ABB RobotStudio station: Practica3.rspag

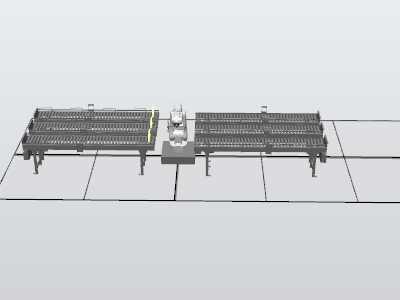
--- station ---
Station Practica3 (saved by RobotStudio 25.4.11475.0)
Controller IRB120_3_58
  mechanical unit ROB_1: IRB120_3_58__01, 6 joints, base frame (0, 0, 0) mm
Layout (positions relative to the parent item):
  - IRB120_3_58__01 [mechanism, from %ABB.RobotStudio.Models.IRB120%\IRB120_3_58_G_01.rslib] at (0, 0, 0) mm; joint values [0, 0, 0, 0, 0.5236, 0] (rad or m)
  - MyNewTool [mechanism] at (364.35, 0, 594) mm, rotated rx -150 ry 0 rz 90 deg
      TCP Centro at (0, 0, 0) mm, rotated rx -90 ry 0 rz 90 deg
      TCP Ventosas3 at (0, 0, -95) mm, rotated rx -90 ry 0 rz 90 deg
      TCP Ventosas4 at (0, 0, 95) mm, rotated rx -90 ry 0 rz 90 deg
      links: Enganche_4
  - Peana [part] at (-200, -200, 0) mm, size 400 x 400 x 100 mm
  - Cinta1 [part] at (-211.15, -1753.75, 0) mm, rotated rx 0 ry 0 rz 90 deg, size 1516.5 x 295 x 472.5 mm
  - Cinta4 [part] at (-387.39, 1694.43, 0) mm, rotated rx 0 ry 0 rz -90 deg, size 1516.5 x 295 x 472.5 mm
  - Cinta2 [part] at (105.68, -1750.96, 0) mm, rotated rx 0 ry 0 rz 90 deg, size 1516.5 x 295 x 472.5 mm
  - Cinta3 [part] at (438.1, -1753.58, 0) mm, rotated rx 0 ry 0 rz 90 deg, size 1516.5 x 295 x 472.5 mm
  - Cinta6 [part] at (250.29, 1696.68, 0) mm, rotated rx 0 ry 0 rz -90 deg, size 1516.5 x 295 x 472.5 mm
  - Cinta5 [part] at (-84.57, 1695.15, 0) mm, rotated rx 0 ry 0 rz -90 deg, size 1516.5 x 295 x 472.5 mm
  - Caja_Tipo1 [part] at (-366, -1693, 382) mm, size 100 x 100 x 50 mm
  - Caja_Tipo2 [part] at (-37, -1686.06, 382.65) mm, size 100 x 100 x 80 mm
  - Caja_Tipo3 [part] at (290, -1683, 388) mm, size 100 x 100 x 100 mm
  - SC_Cinta1 [smart component]
      signals: DI DI_Gen_T1, DI DI_Gen_T2, DI DI_Gen_T3, DO DO_Sensor_Bajo, DO DO_Sensor_Medio, DO DO_Sensor_Alto, DI DI_Mover_C1
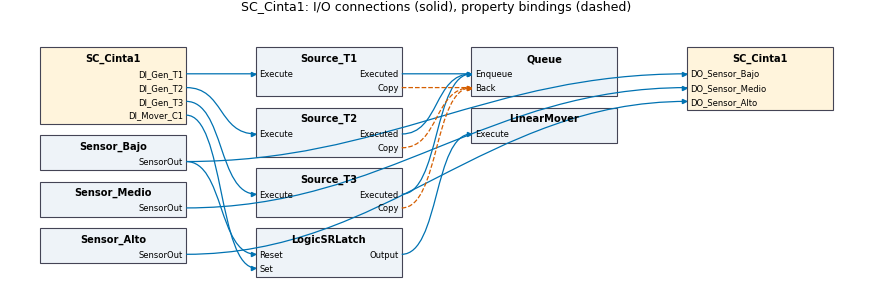
      connections:
        SC_Cinta1.DI_Gen_T1 -> Source_T1.Execute
        SC_Cinta1.DI_Gen_T2 -> Source_T2.Execute
        SC_Cinta1.DI_Gen_T3 -> Source_T3.Execute
        Source_T1.Executed -> Queue.Enqueue
        Source_T2.Executed -> Queue.Enqueue
        Source_T3.Executed -> Queue.Enqueue
        Sensor_Bajo.SensorOut -> SC_Cinta1.DO_Sensor_Bajo
        Sensor_Medio.SensorOut -> SC_Cinta1.DO_Sensor_Medio
        Sensor_Alto.SensorOut -> SC_Cinta1.DO_Sensor_Alto
        Sensor_Bajo.SensorOut -> LogicSRLatch.Reset
        LogicSRLatch.Output -> LinearMover.Execute
        SC_Cinta1.DI_Mover_C1 -> LogicSRLatch.Set
        Source_T1.Copy => Queue.Back
        Source_T2.Copy => Queue.Back
        Source_T3.Copy => Queue.Back
    - Source_T1 [smart component, from Components\Source.rslib] at (0, 878.4, 0) mm
        properties: Source=Caja_Tipo1; Copy=(none); Parent=(none); Position=[-0.366 -1.693 0.382]; Orientation=[0 0 0]; Transient=false; PhysicsBehavior=-1
    - Source_T2 [smart component, from Components\Source.rslib]
        properties: Source=Caja_Tipo2; Copy=(none); Parent=(none); Position=[-0.366 -1.693 0.382]; Orientation=[0 0 0]; Transient=false; PhysicsBehavior=-1
    - Source_T3 [smart component, from Components\Source.rslib]
        properties: Source=Caja_Tipo3; Copy=(none); Parent=(none); Position=[-0.366 -1.693 0.382]; Orientation=[0 0 0]; Transient=false; PhysicsBehavior=-1
    - Queue [smart component, from Components\Queue.rslib]
        properties: Back=(none); Front=(none); Queue={ae4d30b3-6302-4111-9fee-83a94bcd6a61};{9fa5510e-041f-4493-96ec-c95941a7de32};{5319e2fc-a695-4427-a68f-7cbe0e69f7e4};{3efef574-f5d8-49aa-a5b4-01e6362c16f4};{a1e64e2e-bae4-4094-9af5-35717dc52df0};{90407918-cd8a-43af-9253-99db0ca8b2cd};{5acc8fc2-0798-4915-81ff-b25f6d5593ec};{61423d0f-f941-4e73-af3b-112a04a09b53};{953f87a9-bdd4-4cb4-a80c-3d35c462e832};{1631f3d6-8d09-4da0-8cec-8cbaa0fb8792};{cab1151d-17ff-416b-9bb8-76c1a92ffb11};{709a4bb6-f8ae-485e-a46f-52f42bc28a03};{757c1d3f-b98b-4062-b6e4-9dd61a946051};{b9655f3a-bf60-4423-91ba-6a07460e28c4};{d7396197-064d-4214-b519-df7028a49eeb};{af7f2dd8-8d2d-49ce-bc3f-f1ae0ce77ebb};{56c8aa57-b622-4854-bfd4-cc37ea0eaac4};{93e1c836-db4d-4383-b321-3c540578f93f};{c1cab4d0-5605-4614-acff-7234784f2794};{21a5687b-13b3-45a7-a44d-9ef329473538};{e8432f60-373c-4531-8b0a-4d6747e82efe};{1b8eaf30-fe4c-4f09-99cb-c14138031cc8};{9ef8b087-f2a4-45a1-916a-8d388a000a67};{ac3eefbd-dbbd-4806-b8d9-2bdfa1e66709};{6bbb20f7-4848-4c6b-80bb-41a8ed0c3422};{560186ce-d231-4b2f-9cb0-d667fd014fff};{8ef24d2c-7559-482c-9b53-3d872e96b759};{638ee7c7-692f-400c-862d-77c483a76bbb};{18bf07ff-95d7-44c5-ac93-6077ee389aad};{a14bbcad-93fe-4a17-8c33-dc9a6455d2bc};{1956f7e1-81a8-4c4b-a953-4b234403df65};{055c1d69-0d71-46b2-a09d-feb5f3c0ad83};{6400679a-db5a-4c21-bd62-84ae49f8a382};{37c3a838-eb8e-4eb3-96b1-78701e28feef};{289cf7f1-5e36-4ccd-ab18-b29cd6d78d4d};{62f60689-158a-485b-9bfe-8d9deff740b5};{17fe60c0-212e-4ef7-aef1-3c5e78d04126};{c8c3b35f-117b-4ef3-ac39-44fc0f9ecd59};{6bfb9224-18d2-413a-84f5-a1e35e777d4f};{ea2980e8-0bc9-4d52-a2a1-1e1a2d485450};{6993df89-24a9-4713-b949-d7ca80afb984};{2c206039-b06b-44be-9fb2-e4e3ab796f06};{47dba929-5f9b-4cf8-b146-fed9fac773aa};{4920f1fd-ca38-4464-85c7-93d89a30eeed}; NumberOfObjects=2
    - LinearMover [smart component, from Components\LinearMover.rslib]
        properties: Object=Queue; Direction=[0 0.001 0]; Speed=0.15; Reference=Global; ReferenceObject=(none)
    - Sensor_Bajo [smart component, from Components\LineSensor.rslib]
        properties: Start=[-0.411 -0.319 0.42]; End=[-0.21 -0.319 0.42]; Length=0.201; Radius=0; Tag=(none); SenseMultiple=false; SensedPart=(none); SensedPoint=[0 0 0]
      - _sensorPart_ [part], size 201 x 0 x 0 mm
    - Sensor_Medio [smart component, from Components\LineSensor.rslib]
        properties: Start=[-0.411 -0.319 0.46]; End=[-0.21 -0.319 0.46]; Length=0.201; Radius=0; Tag=(none); SenseMultiple=false; SensedPart=(none); SensedPoint=[0 0 0]
      - _sensorPart_ [part], size 201 x 0 x 0 mm
    - Sensor_Alto [smart component, from Components\LineSensor.rslib]
        properties: Start=[-0.411 -0.319 0.48]; End=[-0.21 -0.319 0.48]; Length=0.201; Radius=0; Tag=(none); SenseMultiple=false; SensedPart=(none); SensedPoint=[0 0 0]
      - _sensorPart_ [part], size 201 x 0 x 0 mm
    - LogicSRLatch [smart component, from Components\LogicSRLatch.rslib]
  - SC_Cinta2 [smart component]
      signals: DI DI_Mover_C2, DI DI_Gen_C1, DI DI_Gen_C2, DI DI_Gen_C3, DO DO_Sensor_Bajo, DO DO_Sensor_Medio, DO DO_Sensor_Alto
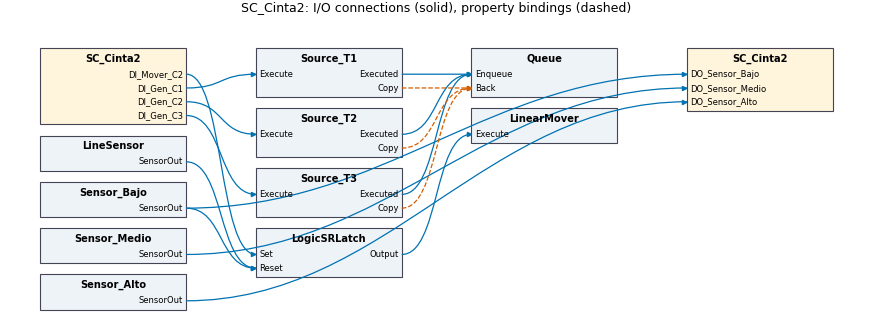
      connections:
        SC_Cinta2.DI_Mover_C2 -> LogicSRLatch.Set
        SC_Cinta2.DI_Gen_C1 -> Source_T1.Execute
        SC_Cinta2.DI_Gen_C2 -> Source_T2.Execute
        SC_Cinta2.DI_Gen_C3 -> Source_T3.Execute
        Source_T1.Executed -> Queue.Enqueue
        Source_T2.Executed -> Queue.Enqueue
        Source_T3.Executed -> Queue.Enqueue
        LogicSRLatch.Output -> LinearMover.Execute
        LineSensor.SensorOut -> LogicSRLatch.Reset
        Sensor_Bajo.SensorOut -> LogicSRLatch.Reset
        Sensor_Bajo.SensorOut -> SC_Cinta2.DO_Sensor_Bajo
        Sensor_Medio.SensorOut -> SC_Cinta2.DO_Sensor_Medio
        Sensor_Alto.SensorOut -> SC_Cinta2.DO_Sensor_Alto
        Source_T3.Copy => Queue.Back
        Source_T2.Copy => Queue.Back
        Source_T1.Copy => Queue.Back
    - LinearMover [smart component, from Components\LinearMover.rslib]
        properties: Object=Queue; Direction=[0 0.001 0]; Speed=0.15; Reference=Global; ReferenceObject=(none)
    - LogicSRLatch [smart component, from Components\LogicSRLatch.rslib]
    - Source_T2 [smart component, from Components\Source.rslib] at (0, 878.4, 0) mm
        properties: Source=Caja_Tipo2; Copy=(none); Parent=(none); Position=[-0.037 -1.683 0.388]; Orientation=[0 0 0]; Transient=false; PhysicsBehavior=-1
    - Source_T3 [smart component, from Components\Source.rslib] at (0, 878.4, 0) mm
        properties: Source=Caja_Tipo3; Copy=(none); Parent=(none); Position=[-0.037 -1.683 0.388]; Orientation=[0 0 0]; Transient=false; PhysicsBehavior=-1
    - Source_T1 [smart component, from Components\Source.rslib] at (0, 878.4, 0) mm
        properties: Source=Caja_Tipo1; Copy=(none); Parent=(none); Position=[-0.037 -1.683 0.388]; Orientation=[0 0 0]; Transient=false; PhysicsBehavior=-1
    - Queue [smart component, from Components\Queue.rslib]
        properties: Back=(none); Front=(none); Queue={2bcd5c23-c1ed-46e9-8c09-8f83fa8b4f7f};{6c76dee3-31f3-442e-bd1e-8fd0cd5ca1d8};{87979af6-ae82-445d-8c1c-a2b879dac4d6};{eee5c5c7-d8e7-4388-a9cb-2509ca800b36};{0ed9a9c4-d81e-4250-8c3f-7bd06b761d9a};{48cb68ef-0ffe-479b-be93-44ded6a24c72};{ede27b09-c003-47f3-a151-95e2712a7b0c};{a391c974-7157-4c51-ac27-7ab25ebc9bf4};{96269cb6-2ddd-45c1-a0d0-c3bba03121e4};{308577e6-806f-4c99-832e-8584b715af30};{7a8da34a-d222-4c7e-9417-0fb4f6fe10c3};{51fd84be-2d47-4bb8-9c48-63eea8f1a314};{4f8447d2-d18b-4198-b70f-0fde71820eac};{26466b57-75da-4393-8d5b-4afc74e56a4b};{388f5636-77e2-470e-ac11-c912e79f43ad};{6e4eb306-18d5-49c2-bef4-ace6f9cce639};{bbdeb09b-5027-4537-9290-c9dec0b41319};{d1ec0450-83df-4b2e-a66f-ffe360aa7048};{c7e78e88-61bb-4ac1-b0f7-c37af5dace11};{622ee8d1-b9ad-42ff-9941-53bfff9b80b7};{5b86faa8-1afa-4e94-a375-27763fc04b84};{0319b542-081c-49c6-b7df-58ec952c4440}; NumberOfObjects=2
    - Sensor_Bajo [smart component, from Components\LineSensor.rslib]
        properties: Start=[-0.085 -0.319 0.42]; End=[0.09 -0.319 0.42]; Length=0.175; Radius=0; Tag=(none); SenseMultiple=false; SensedPart=(none); SensedPoint=[0 0 0]
      - _sensorPart_ [part], size 175 x 0 x 0 mm
    - Sensor_Medio [smart component, from Components\LineSensor.rslib]
        properties: Start=[-0.085 -0.319 0.46]; End=[0.09 -0.319 0.46]; Length=0.175; Radius=0; Tag=(none); SenseMultiple=false; SensedPart=(none); SensedPoint=[0 0 0]
      - _sensorPart_ [part], size 175 x 0 x 0 mm
    - Sensor_Alto [smart component, from Components\LineSensor.rslib]
        properties: Start=[-0.085 -0.319 0.48]; End=[0.09 -0.319 0.48]; Length=0.175; Radius=0; Tag=(none); SenseMultiple=false; SensedPart=(none); SensedPoint=[0 0 0]
      - _sensorPart_ [part], size 175 x 0 x 0 mm
  - SC_Cinta3 [smart component]
      signals: DI DI_Gen_T1, DI DI_Gen_T2, DI DI_Gen_T3, DO DO_Sensor_Bajo, DO DO_Sensor_Medio, DO DO_Sensor_Alto, DI DI_Mover_C3
      connections:
        LogicSRLatch_3.Output -> LinearMover_2.Execute
        Source_T1.Executed -> Queue_2.Enqueue
        Source_T2.Executed -> Queue_2.Enqueue
        Source_T3.Executed -> Queue_2.Enqueue
        SC_Cinta3.DI_Gen_T1 -> Source_T1.Execute
        SC_Cinta3.DI_Gen_T2 -> Source_T2.Execute
        SC_Cinta3.DI_Gen_T3 -> Source_T3.Execute
        Sensor_Bajo.SensorOut -> SC_Cinta3.DO_Sensor_Bajo
        Sensor_Bajo.SensorOut -> LogicSRLatch_3.Reset
        Sensor_Medio.SensorOut -> SC_Cinta3.DO_Sensor_Medio
        Sensor_Alto.SensorOut -> SC_Cinta3.DO_Sensor_Alto
        SC_Cinta3.DI_Mover_C3 -> LogicSRLatch_3.Set
        Source_T1.Copy => Queue_2.Back
        Source_T2.Copy => Queue_2.Back
        Source_T3.Copy => Queue_2.Back
    - Source_T1 [smart component, from Components\Source.rslib]
        properties: Source=Caja_Tipo1; Copy=(none); Parent=(none); Position=[0.29 -1.683 0.388]; Orientation=[0 0 0]; Transient=false; PhysicsBehavior=-1
    - Sensor_Bajo [smart component, from Components\LineSensor.rslib]
        properties: Start=[0.237 -0.319 0.42]; End=[0.438 -0.319 0.42]; Length=0.201; Radius=0; Tag=(none); SenseMultiple=false; SensedPart=(none); SensedPoint=[0 0 0]
      - _sensorPart_ [part], size 201 x 0 x 0 mm
    - Queue_2 [smart component, from Components\Queue.rslib]
        properties: Back=(none); Front=(none); Queue={b5c0da53-b886-4eab-a8f7-240ca8277bb4};{162bf9dd-af30-44ee-bf84-297d0a330099};{1ce0c98b-bb50-4a90-8f2b-f630c16990df};{7d84dcbd-445a-4615-af1b-5e8ef1b0da41};{f2ce0fef-d506-4055-bce7-edc570f5b85d};{49ed6fa6-4484-4528-a036-6e04abb92bae};{51e9f9c3-66fc-43a1-92ef-84e0ce0dd9ee};{a6f4487b-d18e-4f28-a26b-d157c1f4e47e};{40463528-f2a5-4b0f-801e-c86bb77c77c6};{7bbab9be-23ff-4f72-bedf-08c0365cb3c3};{96a9fc0c-d42f-4625-b4ce-ff104d0d23d5};{38a37ed4-7e6c-411f-af4e-19aff20a759d};{77cec95b-3a46-431e-99ce-bad3b8b5176a};{a7fffe4b-cb80-4798-9ffc-81a953cfccc9};{07ba421a-4e5e-4a4c-8141-2298dd789c99};{14acecfe-8c89-4afa-883c-57a0848518f5};{03d718bc-ab0b-4980-ad5a-f10c83bcab31};{af4d491e-c72f-4645-8bd7-c3d7c8b11cec};{0fcde2d3-d7fc-49db-9a2c-edd93dbc6e02};{0f9b7fda-dccf-447b-aa29-b1cebfc17353};{32b10893-1c7e-43b2-a21f-2af3cf555bbd};{ef222544-086f-4277-904e-25c3415c13a1};{819d3b9b-c1dd-4f60-9c29-6154756c0372};{19730fc8-a8c3-4879-83ee-9a8b8ef66b87};{472fec01-8044-440c-8fff-ca474cbc4876};{4a0d8dfd-107d-4185-9536-f8a48dfdc9b6};{2941b239-3e65-4e98-8b67-6c5e40cb0733}; NumberOfObjects=1
    - LinearMover_2 [smart component, from Components\LinearMover.rslib]
        properties: Object=Queue_2; Direction=[0 0.001 0]; Speed=0.15; Reference=Global; ReferenceObject=(none)
    - LogicSRLatch_3 [smart component, from Components\LogicSRLatch.rslib]
    - Source_T2 [smart component, from Components\Source.rslib]
        properties: Source=Caja_Tipo2; Copy=(none); Parent=(none); Position=[0.29 -1.683 0.388]; Orientation=[0 0 0]; Transient=false; PhysicsBehavior=-1
    - Source_T3 [smart component, from Components\Source.rslib]
        properties: Source=Caja_Tipo3; Copy=(none); Parent=(none); Position=[0.29 -1.683 0.388]; Orientation=[0 0 0]; Transient=false; PhysicsBehavior=-1
    - Sensor_Medio [smart component, from Components\LineSensor.rslib]
        properties: Start=[0.237 -0.319 0.46]; End=[0.438 -0.319 0.46]; Length=0.201; Radius=0; Tag=(none); SenseMultiple=false; SensedPart=(none); SensedPoint=[0 0 0]
      - _sensorPart_ [part], size 201 x 0 x 0 mm
    - Sensor_Alto [smart component, from Components\LineSensor.rslib]
        properties: Start=[0.237 -0.319 0.48]; End=[0.438 -0.319 0.48]; Length=0.201; Radius=0; Tag=(none); SenseMultiple=false; SensedPart=(none); SensedPoint=[0 0 0]
      - _sensorPart_ [part], size 201 x 0 x 0 mm
  - SC_Agarre [smart component]
      connections:
        LogicGate.Output -> Detacher.Execute
        CollisionSensor_2.SensorOut -> Detacher.Execute
        CollisionSensor.SensorOut -> Attacher.Execute
        CollisionSensor_3.SensorOut -> Attacher_2.Execute
        CollisionSensor_4.SensorOut -> Detacher_2.Execute
        CollisionSensor_2.SensorOut -> Detacher_2.Execute
        CollisionSensor.Part2 => Attacher.Child
        CollisionSensor.Part2 => Detacher.Child
        CollisionSensor_3.Part2 => Attacher_2.Child
        CollisionSensor_3.Part2 => Detacher.Child
    - Attacher [smart component, from Components\Attacher.rslib]
        properties: Parent=MyNewTool; Flange=1; Child=(none); Mount=false; Offset=[0 0 0]; Orientation=[0 0 0]
    - Detacher [smart component, from Components\Detacher.rslib]
        properties: Child=(none); KeepPosition=true
    - CollisionSensor [smart component, from Components\CollisionSensor.rslib]
        properties: Object1=MyNewTool; Object2=(none); NearMiss=0; Part1=(none); Part2=(none); CollisionType=0
    - CollisionSensor_2 [smart component, from Components\CollisionSensor.rslib]
        properties: Object1=MyNewTool; Object2=Grupo_1; NearMiss=0; Part1=(none); Part2=(none); CollisionType=0
    - CollisionSensor_3 [smart component, from Components\CollisionSensor.rslib]
        properties: Object1=MyNewTool; Object2=(none); NearMiss=0; Part1=(none); Part2=(none); CollisionType=0
    - Attacher_2 [smart component, from Components\Attacher.rslib]
        properties: Parent=MyNewTool; Flange=2; Child=(none); Mount=false; Offset=[0 0 0]; Orientation=[0 0 0]
  - Grupo_1 [graphiccomponentgroup]
    - Caja [part] at (-339.08, 251.28, 364.37) mm, size 100 x 100 x 50 mm
    - Caja_2 [part] at (-37, 355.02, 378.78) mm, size 100 x 100 x 80 mm
    - Pieza_1 [part] at (37.54, -45.56, 52.42) mm, size 100 x 100 x 100 mm
Attachment: MyNewTool is attached to IRB120_3_58__01 / Link6
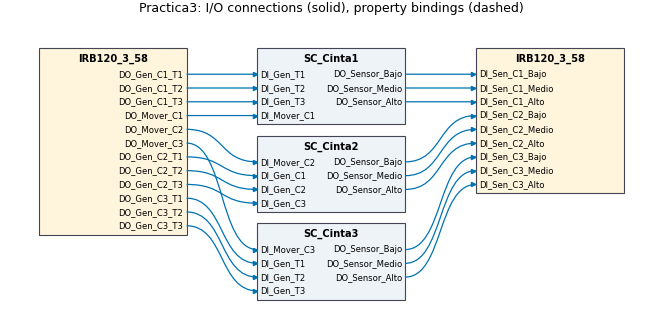
Station logic (signal -> signal, property => property):
  IRB120_3_58.DO_Gen_C1_T1 -> SC_Cinta1.DI_Gen_T1
  IRB120_3_58.DO_Gen_C1_T2 -> SC_Cinta1.DI_Gen_T2
  IRB120_3_58.DO_Gen_C1_T3 -> SC_Cinta1.DI_Gen_T3
  SC_Cinta1.DO_Sensor_Bajo -> IRB120_3_58.DI_Sen_C1_Bajo
  SC_Cinta1.DO_Sensor_Medio -> IRB120_3_58.DI_Sen_C1_Medio
  SC_Cinta1.DO_Sensor_Alto -> IRB120_3_58.DI_Sen_C1_Alto
  IRB120_3_58.DO_Mover_C1 -> SC_Cinta1.DI_Mover_C1
  IRB120_3_58.DO_Mover_C2 -> SC_Cinta2.DI_Mover_C2
  IRB120_3_58.DO_Mover_C3 -> SC_Cinta3.DI_Mover_C3
  SC_Cinta2.DO_Sensor_Bajo -> IRB120_3_58.DI_Sen_C2_Bajo
  SC_Cinta2.DO_Sensor_Medio -> IRB120_3_58.DI_Sen_C2_Medio
  SC_Cinta2.DO_Sensor_Alto -> IRB120_3_58.DI_Sen_C2_Alto
  SC_Cinta3.DO_Sensor_Bajo -> IRB120_3_58.DI_Sen_C3_Bajo
  SC_Cinta3.DO_Sensor_Medio -> IRB120_3_58.DI_Sen_C3_Medio
  SC_Cinta3.DO_Sensor_Alto -> IRB120_3_58.DI_Sen_C3_Alto
  IRB120_3_58.DO_Gen_C2_T1 -> SC_Cinta2.DI_Gen_C1
  IRB120_3_58.DO_Gen_C2_T2 -> SC_Cinta2.DI_Gen_C2
  IRB120_3_58.DO_Gen_C2_T3 -> SC_Cinta2.DI_Gen_C3
  IRB120_3_58.DO_Gen_C3_T1 -> SC_Cinta3.DI_Gen_T1
  IRB120_3_58.DO_Gen_C3_T2 -> SC_Cinta3.DI_Gen_T2
  IRB120_3_58.DO_Gen_C3_T3 -> SC_Cinta3.DI_Gen_T3

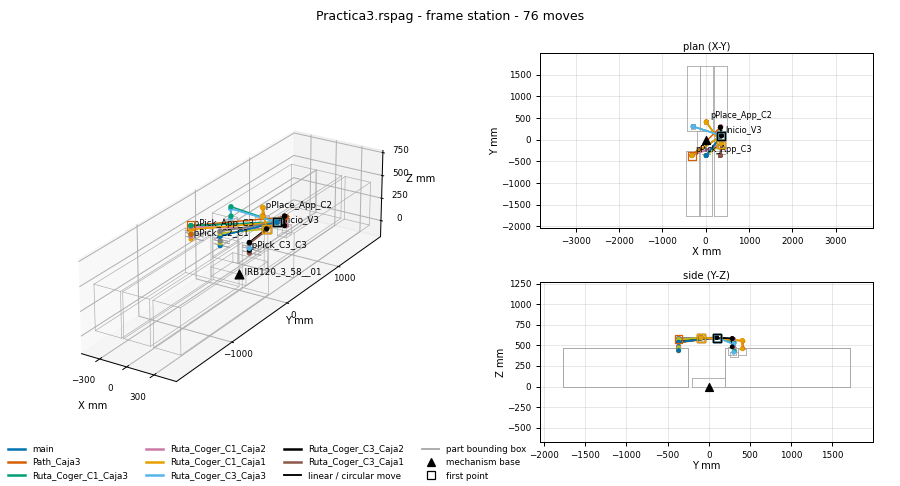
[picture p0: tool path of Practica3.rspag in frame station, 76 of 76 moves have a stored position in this frame; points joined in program order, loops and branches not executed]
--- Controller Data/IRB120_3_58/RAPID/TASK1/PROGMOD/CalibData.mod ---
MODULE CalibData
    PERS tooldata Centro:=[TRUE,[[0,0,0],[1,0,0,0]],[1,[0,0,1],[1,0,0,0],0,0,0]];
    PERS tooldata Ventosas3:=[TRUE,[[0,95,0],[1,0,0,0]],[1,[0,0,1],[1,0,0,0],0,0,0]];
    PERS tooldata Ventosas4:=[TRUE,[[0,-95,0],[1,0,0,0]],[1,[0,0,1],[1,0,0,0],0,0,0]];
ENDMODULE

--- Controller Data/IRB120_3_58/RAPID/TASK1/PROGMOD/Module1.mod ---
MODULE Module1


    CONST robtarget pPick_App_C3:=[[-316,-368.6,572],[0,0,-0.707106781,0.707106781],[-2,0,-2,0],[9E+09,9E+09,9E+09,9E+09,9E+09,9E+09]];
    CONST robtarget pPick_C3_C_1:=[[-316,-368.6,482],[0,0,-0.707106781,0.707106781],[-2,1,-3,0],[9E+09,9E+09,9E+09,9E+09,9E+09,9E+09]];
    CONST robtarget pPlace_App_C6:=[[349.296,299.975,572],[0.5,-0.5,0.5,-0.5],[0,-1,-1,0],[9E+09,9E+09,9E+09,9E+09,9E+09,9E+09]];
    CONST robtarget pPlace_C3_C_6:=[[349.296,299.975,482],[0.5,-0.5,0.5,-0.5],[0,-2,0,0],[9E+09,9E+09,9E+09,9E+09,9E+09,9E+09]];
    CONST robtarget Inicio_V3:=[[364.353821314,95.000001192,593.99994615],[0.499999995,0,0.866025407,0],[-1,0,-1,0],[9E+09,9E+09,9E+09,9E+09,9E+09,9E+09]];

    ! Variables para la generacion aleatoria
    VAR num nCintaAleatoria := 0;
    VAR num nTipoAleatorio := 0;
    VAR num nSeed := 42;

    ! Contadores y requeridas
    VAR num nCajasT1_Req := 0;
    VAR num nCajasT2_Req := 0;
    VAR num nCajasT3_Req := 0;
    VAR num nCajasT1_Gen := 0;
    VAR num nCajasT2_Gen := 0;
    VAR num nCajasT3_Gen := 0;
    VAR num nTotalCajas := 0;
    VAR num nCajasProcesadas := 0;
   ! Posición de los diferentes puntos
    CONST robtarget pPick_C3_C1:=[[-316,-368.6,482],[0,0,-0.707106781,0.707106781],[-2,1,-3,0],[9E+09,9E+09,9E+09,9E+09,9E+09,9E+09]];
    CONST robtarget pPlace_App_C3:=[[349.296,299.975,572],[0.5,-0.5,0.5,-0.5],[0,-1,-1,0],[9E+09,9E+09,9E+09,9E+09,9E+09,9E+09]];
    CONST robtarget pPlace_C3:=[[349.296,299.975,482],[0.5,-0.5,0.5,-0.5],[0,-2,0,0],[9E+09,9E+09,9E+09,9E+09,9E+09,9E+09]];
    CONST robtarget Inicio_V4:=[[364.353851784,-95,594.000006911],[0.500000003,0,0.866025402,0],[-1,0,0,0],[9E+09,9E+09,9E+09,9E+09,9E+09,9E+09]];
    CONST robtarget pPick_App_C2:=[[-316.000000141,-368.6,562],[0.707106781,0.707106781,-0.000000001,0],[-2,0,0,0],[9E+09,9E+09,9E+09,9E+09,9E+09,9E+09]];
    CONST robtarget pPick_C2_C1:=[[-316,-368.6,462],[0.707106781,0.707106781,-0.000000001,0],[-2,1,-1,0],[9E+09,9E+09,9E+09,9E+09,9E+09,9E+09]];
    CONST robtarget pPick_App_C1:=[[-315.999999859,-368.6,532],[-0.000000001,0,0.707106781,-0.707106781],[-2,0,-2,0],[9E+09,9E+09,9E+09,9E+09,9E+09,9E+09]];
    CONST robtarget pPick_C1_C1:=[[-316,-368.6,432],[0.000000001,0,-0.707106781,0.707106781],[-2,1,-3,0],[9E+09,9E+09,9E+09,9E+09,9E+09,9E+09]];
    CONST robtarget pPlace_App_C1:=[[-289.15,308.032,532],[0.707106781,-0.707106781,-0.000000002,0.000000002],[1,-1,-1,0],[9E+09,9E+09,9E+09,9E+09,9E+09,9E+09]];
    CONST robtarget pPlace_C1:=[[-289.15,308.032,432],[0.707106781,-0.707106781,-0.000000002,0.000000002],[1,-2,0,0],[9E+09,9E+09,9E+09,9E+09,9E+09,9E+09]];
    CONST robtarget pPlace_App_C2:=[[15.071999873,413.101,552],[0.499999999,0.5,-0.500000001,-0.5],[0,1,0,0],[9E+09,9E+09,9E+09,9E+09,9E+09,9E+09]];
    CONST robtarget pPlace_C2:=[[15.072,413.101,462],[0.499999999,0.5,-0.500000001,-0.5],[0,0,-1,0],[9E+09,9E+09,9E+09,9E+09,9E+09,9E+09]];
    CONST robtarget pPick_App__C3_C3:=[[339.99999988,-365.8,548],[0.500000001,-0.5,0.499999999,-0.5],[-1,0,-2,0],[9E+09,9E+09,9E+09,9E+09,9E+09,9E+09]];
    CONST robtarget pPick_C3_C3:=[[340,-365.8,488],[0.500000001,-0.5,0.499999999,-0.5],[-1,1,-3,0],[9E+09,9E+09,9E+09,9E+09,9E+09,9E+09]];
    CONST robtarget pPick_App_C2_C3:=[[340.00000016,-365.8,548],[0.499999999,0.5,0.500000001,0.5],[-1,0,0,0],[9E+09,9E+09,9E+09,9E+09,9E+09,9E+09]];
    CONST robtarget pPick_C2_C3:=[[340,-365.8,468],[0.499999999,0.5,0.500000001,0.5],[-1,1,-1,0],[9E+09,9E+09,9E+09,9E+09,9E+09,9E+09]];
    CONST robtarget pPick_App_C1_C3:=[[339.999999859,-365.8,538],[0.000000001,0,0.707106781,-0.707106781],[-1,-1,-1,0],[9E+09,9E+09,9E+09,9E+09,9E+09,9E+09]];
    CONST robtarget pPick_C1_C3:=[[340,-365.8,438],[0.000000001,0,0.707106781,-0.707106781],[-1,-2,0,0],[9E+09,9E+09,9E+09,9E+09,9E+09,9E+09]];
    CONST robtarget pPick_App_C3_C_2:=[[13.000012661,-365.800008465,587.999971855],[0.50000001,-0.500000001,0.499999988,-0.500000001],[-2,1,-2,0],[9E+09,9E+09,9E+09,9E+09,9E+09,9E+09]];
    CONST robtarget pPick_C3_C2:=[[13,-365.8,488],[0.500000001,-0.499999999,0.499999999,-0.500000001],[-2,0,-3,0],[9E+09,9E+09,9E+09,9E+09,9E+09,9E+09]];
    CONST robtarget pPick_App_C2_C2:=[[12.9999999,-365.7999999,568],[0.500000001,0.5,0.5,0.5],[-2,1,0,0],[9E+09,9E+09,9E+09,9E+09,9E+09,9E+09]];
    CONST robtarget pPick_C2_C2:=[[13,-365.8,468],[0.500000001,0.5,0.5,0.5],[-2,0,-1,0],[9E+09,9E+09,9E+09,9E+09,9E+09,9E+09]];
    CONST robtarget pPick_App_C1_C2:=[[13.0000002,-365.8,538],[0.5,-0.500000001,0.5,-0.499999999],[-2,1,-2,0],[9E+09,9E+09,9E+09,9E+09,9E+09,9E+09]];
    CONST robtarget pPick_C1_C2:=[[13,-365.8,438],[0.5,-0.500000001,0.5,-0.499999999],[-2,0,-3,0],[9E+09,9E+09,9E+09,9E+09,9E+09,9E+09]];
    CONST robtarget pPlace_App_3:=[[337.838,283.8969998,582.539],[0.500000001,-0.5,0.5,-0.499999999],[0,-1,-1,0],[9E+09,9E+09,9E+09,9E+09,9E+09,9E+09]];
    CONST robtarget pPlace_3:=[[337.838,283.897,482.539],[0.500000001,-0.5,0.5,-0.499999999],[0,-2,0,0],[9E+09,9E+09,9E+09,9E+09,9E+09,9E+09]];
    CONST robtarget pPlace_App_1:=[[-289.081000141,301.279,514.372],[0.707106781,-0.707106781,-0.000000001,0],[1,-2,0,0],[9E+09,9E+09,9E+09,9E+09,9E+09,9E+09]];
    CONST robtarget pPlace_1:=[[-289.081,301.279,414.372],[0.707106781,-0.707106781,-0.000000001,0],[1,-2,0,0],[9E+09,9E+09,9E+09,9E+09,9E+09,9E+09]];
    CONST robtarget pPlace_App_2:=[[12.9999999,405.0210001,558.778],[0.5,0.5,-0.500000001,-0.5],[0,1,0,0],[9E+09,9E+09,9E+09,9E+09,9E+09,9E+09]];
    CONST robtarget pPlace_2:=[[13,405.021,458.778],[0.5,0.5,-0.5,-0.500000001],[0,0,-1,0],[9E+09,9E+09,9E+09,9E+09,9E+09,9E+09]];


    PROC main()

        ! Inicializar variables
        nCajasT1_Gen := 0;
        nCajasT2_Gen := 0;
        nCajasT3_Gen := 0;
        nCajasProcesadas := 0;

        !PEDIR DATOS AL USUARIO EN EL FLEXPENDANT
        TPErase; ! Limpiamos la pantalla
        TPWrite "=====================================";
        TPWrite "   CONFIGURACION DE PRODUCCION";
        TPWrite "=====================================";
        TPReadNum nCajasT1_Req, "Numero de cajas Tipo 1 a generar:";
        TPReadNum nCajasT2_Req, "Numero de cajas Tipo 2 a generar:";
        TPReadNum nCajasT3_Req, "Numero de cajas Tipo 3 a generar:";

        nTotalCajas := nCajasT1_Req + nCajasT2_Req + nCajasT3_Req;

        TPWrite " ";
        TPWrite "-> Produccion Total: " \Num:=nTotalCajas;
        TPWrite "=====================================";
        WaitTime 1.5;

        ! Colocar el robot en su posición inicial
        MoveJ Inicio_V3, v1000, fine, Ventosas3\WObj:=wobj0;

        ! Encender cintas
        SetDO DO_Mover_C1, 1;
        SetDO DO_Mover_C2, 1;
        SetDO DO_Mover_C3, 1;

        WaitTime 1;

        ! BUCLE SECUENCIAL LIMITADO POR CANTIDAD
        WHILE nCajasProcesadas < nTotalCajas DO

            GenerarCajaAleatoria;

            ! Esperar a que la caja llegue a la zona de recogida
            WaitUntil (DI_Sen_C1_Bajo = 1 OR DI_Sen_C2_Bajo = 1 OR DI_Sen_C3_Bajo = 1);
            WaitTime 0.3;

            ! Para las cintas para correcto procesamiento
            SetDO DO_Mover_C1, 0;
            SetDO DO_Mover_C2, 0;
            SetDO DO_Mover_C3, 0;
            WaitTime 0.2;

            ! Procesar la caja
            IF DI_Sen_C1_Bajo = 1 THEN
                IF DI_Sen_C1_Medio = 0 AND DI_Sen_C1_Alto = 0 THEN
                    Ruta_Coger_C1_Caja1; Ruta_Dejar1;
                ELSEIF DI_Sen_C1_Medio = 1 AND DI_Sen_C1_Alto = 0 THEN
                    Ruta_Coger_C1_Caja2; Ruta_Dejar2;
                ELSEIF DI_Sen_C1_Medio = 1 AND DI_Sen_C1_Alto = 1 THEN
                    Ruta_Coger_C1_Caja3; Ruta_Dejar3;
                ENDIF

            ELSEIF DI_Sen_C2_Bajo = 1 THEN
                IF DI_Sen_C2_Medio = 0 AND DI_Sen_C2_Alto = 0 THEN
                    Ruta_Coger_C2_Caja1; Ruta_Dejar1;
                ELSEIF DI_Sen_C2_Medio = 1 AND DI_Sen_C2_Alto = 0 THEN
                    Ruta_Coger_C2_Caja2; Ruta_Dejar2;
                ELSEIF DI_Sen_C2_Medio = 1 AND DI_Sen_C2_Alto = 1 THEN
                    Ruta_Coger_C2_Caja3; Ruta_Dejar3;
                ENDIF

            ELSEIF DI_Sen_C3_Bajo = 1 THEN
                IF DI_Sen_C3_Medio = 0 AND DI_Sen_C3_Alto = 0 THEN
                    Ruta_Coger_C3_Caja1; Ruta_Dejar1;
                ELSEIF DI_Sen_C3_Medio = 1 AND DI_Sen_C3_Alto = 0 THEN
                    Ruta_Coger_C3_Caja2; Ruta_Dejar2;
                ELSEIF DI_Sen_C3_Medio = 1 AND DI_Sen_C3_Alto = 1 THEN
                    Ruta_Coger_C3_Caja3; Ruta_Dejar3;
                ENDIF
            ENDIF

            ! Esperar a que el robot llegue a la posición inicial
            WaitRob \InPos;

            ! Actualizar contador
            nCajasProcesadas := nCajasProcesadas + 1;

            ! Reactivar las cintas de entrada
            SetDO DO_Mover_C1, 1;
            SetDO DO_Mover_C2, 1;
            SetDO DO_Mover_C3, 1;

            WaitTime 0.5;

        ENDWHILE

        ! Mensaje de finalizacion del programa
        TPWrite "=====================================";
        TPWrite "  ¡PRODUCCION COMPLETADA CON EXITO!  ";
        TPWrite "=====================================";
        Stop; ! Detener la ejecución

    ENDPROC

    ! Subrutina para generar cajas aleatorias en cintas aleatorias
    PROC GenerarCajaAleatoria()
        VAR bool bGenerada := FALSE;

        WHILE bGenerada = FALSE DO

            ! Calculo  del LCG para cintas y tipos
            nSeed := (nSeed * 13 + 7) MOD 1000;
            ! Normalizar el numero para las 3 cintas (0, 1 , 2)
            nCintaAleatoria := (nSeed MOD 3) + 1;

            nSeed := (nSeed * 13 + 7) MOD 1000;
            ! Normalizar el numero para los 3 tipos de cajas (0, 1 , 2)
            nTipoAleatorio := (nSeed MOD 3) + 1;

            ! Comprobar si se ha pedido esa caja y generar la caja requerida
            IF nTipoAleatorio = 1 AND nCajasT1_Gen < nCajasT1_Req THEN
                IF nCintaAleatoria = 1 THEN PulseDO \PLength:=0.02, DO_Gen_C1_T1;
                ELSEIF nCintaAleatoria = 2 THEN PulseDO \PLength:=0.02, DO_Gen_C2_T1;
                ELSEIF nCintaAleatoria = 3 THEN PulseDO \PLength:=0.02, DO_Gen_C3_T1; ENDIF

                nCajasT1_Gen := nCajasT1_Gen + 1;
                TPWrite ">>> Generada TIPO 1 en Cinta " \Num:=nCintaAleatoria;
                bGenerada := TRUE;

            ELSEIF nTipoAleatorio = 2 AND nCajasT2_Gen < nCajasT2_Req THEN
                IF nCintaAleatoria = 1 THEN PulseDO \PLength:=0.02, DO_Gen_C1_T2;
                ELSEIF nCintaAleatoria = 2 THEN PulseDO \PLength:=0.02, DO_Gen_C2_T2;
                ELSEIF nCintaAleatoria = 3 THEN PulseDO \PLength:=0.02, DO_Gen_C3_T2; ENDIF

                nCajasT2_Gen := nCajasT2_Gen + 1;
                TPWrite ">>> Generada TIPO 2 en Cinta " \Num:=nCintaAleatoria;
                bGenerada := TRUE;

            ELSEIF nTipoAleatorio = 3 AND nCajasT3_Gen < nCajasT3_Req THEN
                IF nCintaAleatoria = 1 THEN PulseDO \PLength:=0.02, DO_Gen_C1_T3;
                ELSEIF nCintaAleatoria = 2 THEN PulseDO \PLength:=0.02, DO_Gen_C2_T3;
                ELSEIF nCintaAleatoria = 3 THEN PulseDO \PLength:=0.02, DO_Gen_C3_T3; ENDIF

                nCajasT3_Gen := nCajasT3_Gen + 1;
                TPWrite ">>> Generada TIPO 3 en Cinta " \Num:=nCintaAleatoria;
                bGenerada := TRUE;
            ENDIF

            ! Si el tipo elegido al azar ya había llegado a su límite de cajas,
            ! el bucle WHILE repetirá el proceso milisegundos después buscando
            ! otro tipo que aún necesitemos crear.

        ENDWHILE
    ENDPROC

! Trayectorias del robot
    PROC Path_Caja3()
        MoveL pPick_App_C3,v1000,fine,Ventosas3\WObj:=wobj0;
        MoveL pPick_C3_C_1,v1000,fine,Ventosas3\WObj:=wobj0;
        MoveL pPick_App_C3,v1000,fine,Ventosas3\WObj:=wobj0;
        MoveL pPlace_App_C6,v1000,z100,Ventosas3\WObj:=wobj0;
        MoveL pPlace_C3_C_6,v1000,fine,Ventosas3\WObj:=wobj0;
        MoveL pPlace_App_C6,v1000,fine,Ventosas3\WObj:=wobj0;
    ENDPROC
    PROC Ruta_Coger_C1_Caja3()
        MoveL Inicio_V3,v1000,fine,Ventosas3\WObj:=wobj0;
        MoveL pPick_App_C3,v1000,fine,Ventosas3\WObj:=wobj0;
        MoveL pPick_C3_C1,v1000,fine,Ventosas3\WObj:=wobj0;
        MoveL pPick_App_C3,v1000,fine,Ventosas3\WObj:=wobj0;
        MoveL Inicio_V3,v1000,fine,Ventosas3\WObj:=wobj0;
    ENDPROC
    PROC Ruta_Coger_C1_Caja2()
        MoveL Inicio_V4,v500,fine,Ventosas4\WObj:=wobj0;
        MoveL pPick_App_C2,v1000,fine,Ventosas4\WObj:=wobj0;
        MoveL pPick_C2_C1,v1000,fine,Ventosas4\WObj:=wobj0;
        MoveL pPick_App_C2,v1000,fine,Ventosas4\WObj:=wobj0;
        MoveL Inicio_V4,v1000,fine,Ventosas4\WObj:=wobj0;
    ENDPROC
    PROC Ruta_Coger_C1_Caja1()
        MoveL Inicio_V3,v1000,fine,Ventosas3\WObj:=wobj0;
        MoveL pPick_App_C1,v1000,fine,Ventosas3\WObj:=wobj0;
        MoveL pPick_C1_C1,v1000,fine,Ventosas3\WObj:=wobj0;
        MoveL pPick_App_C1,v1000,fine,Ventosas3\WObj:=wobj0;
        MoveL Inicio_V3,v1000,fine,Ventosas3\WObj:=wobj0;
    ENDPROC
    PROC Ruta_Coger_C3_Caja3()
        MoveL Inicio_V3,v1000,fine,Ventosas3\WObj:=wobj0;
        MoveL pPick_App__C3_C3,v1000,fine,Ventosas3\WObj:=wobj0;
        MoveL pPick_C3_C3,v1000,fine,Ventosas3\WObj:=wobj0;
        MoveL pPick_App__C3_C3,v1000,fine,Ventosas3\WObj:=wobj0;
        MoveL Inicio_V3,v1000,fine,Ventosas3\WObj:=wobj0;
    ENDPROC
    PROC Ruta_Coger_C3_Caja2()
        MoveL Inicio_V4,v1000,fine,Ventosas4\WObj:=wobj0;
        MoveL pPick_App_C2_C3,v1000,fine,Ventosas4\WObj:=wobj0;
        MoveL pPick_C2_C3,v1000,fine,Ventosas4\WObj:=wobj0;
        MoveL pPick_App_C2_C3,v1000,fine,Ventosas4\WObj:=wobj0;
        MoveL Inicio_V4,v1000,fine,Ventosas4\WObj:=wobj0;
    ENDPROC
    PROC Ruta_Coger_C3_Caja1()
        MoveL Inicio_V3,v1000,fine,Ventosas3\WObj:=wobj0;
        MoveL pPick_App_C1_C3,v1000,fine,Ventosas3\WObj:=wobj0;
        MoveL pPick_C1_C3,v1000,fine,Ventosas3\WObj:=wobj0;
        MoveL pPick_App_C1_C3,v1000,fine,Ventosas3\WObj:=wobj0;
        MoveL Inicio_V3,v1000,fine,Ventosas3\WObj:=wobj0;
    ENDPROC
    PROC Ruta_Coger_C2_Caja3()
        MoveL Inicio_V3,v1000,fine,Ventosas3\WObj:=wobj0;
        MoveL pPick_App_C3_C_2,v1000,fine,Ventosas3\WObj:=wobj0;
        MoveL pPick_C3_C2,v1000,fine,Ventosas3\WObj:=wobj0;
        MoveL pPick_App_C3_C_2,v1000,fine,Ventosas3\WObj:=wobj0;
        MoveL Inicio_V3,v1000,fine,Ventosas3\WObj:=wobj0;
    ENDPROC
    PROC Ruta_Coger_C2_Caja2()
        MoveL Inicio_V4,v1000,fine,Ventosas4\WObj:=wobj0;
        MoveL pPick_App_C2_C2,v1000,fine,Ventosas4\WObj:=wobj0;
        MoveL pPick_C2_C2,v1000,fine,Ventosas4\WObj:=wobj0;
        MoveL pPick_App_C2_C2,v1000,fine,Ventosas4\WObj:=wobj0;
        MoveL Inicio_V4,v1000,fine,Ventosas4\WObj:=wobj0;
    ENDPROC
    PROC Ruta_Coger_C2_Caja1()
        MoveL Inicio_V3,v1000,fine,Ventosas3\WObj:=wobj0;
        MoveL pPick_App_C1_C2,v1000,fine,Ventosas3\WObj:=wobj0;
        MoveL pPick_C1_C2,v1000,fine,Ventosas3\WObj:=wobj0;
        MoveL pPick_App_C1_C2,v1000,fine,Ventosas3\WObj:=wobj0;
        MoveL Inicio_V3,v1000,fine,Ventosas3\WObj:=wobj0;
    ENDPROC
    PROC Caja2()
        MoveL Inicio_V4,v1000,z100,Ventosas4\WObj:=wobj0;
        MoveL pPlace_App_C2,v1000,z100,Ventosas4\WObj:=wobj0;
        MoveL pPlace_C2,v1000,z100,Ventosas4\WObj:=wobj0;
    ENDPROC
    PROC Caja1()
        MoveL Inicio_V3,v1000,z100,Ventosas3\WObj:=wobj0;
        MoveL pPlace_App_C1,v1000,z100,Ventosas3\WObj:=wobj0;
        MoveL pPlace_C1,v1000,z100,Ventosas3\WObj:=wobj0;
    ENDPROC
    PROC Caja3()
        MoveL Inicio_V3,v1000,z100,Ventosas3\WObj:=wobj0;
        MoveL pPlace_App_C3,v1000,z100,Ventosas3\WObj:=wobj0;
        MoveL pPlace_C3,v1000,z100,Ventosas3\WObj:=wobj0;
   ENDPROC
    PROC Ruta_Dejar2()
        MoveL Inicio_V4,v1000,fine,Ventosas4\WObj:=wobj0;
        MoveL pPlace_App_2,v1000,fine,Ventosas4\WObj:=wobj0;
        MoveL pPlace_2,v1000,fine,Ventosas4\WObj:=wobj0;
        MoveL pPlace_App_2,v1000,fine,Ventosas4\WObj:=wobj0;
        MoveL Inicio_V4,v1000,fine,Ventosas4\WObj:=wobj0;
    ENDPROC
    PROC Ruta_Dejar1()
        MoveL Inicio_V3,v1000,fine,Ventosas3\WObj:=wobj0;
        MoveL pPlace_App_1,v1000,fine,Ventosas3\WObj:=wobj0;
        MoveL pPlace_1,v1000,fine,Ventosas3\WObj:=wobj0;
        MoveL pPlace_App_1,v1000,fine,Ventosas3\WObj:=wobj0;
        MoveL Inicio_V3,v1000,fine,Ventosas3\WObj:=wobj0;
    ENDPROC
    PROC Ruta_Dejar3()
        MoveL Inicio_V3,v1000,fine,Ventosas3\WObj:=wobj0;
        MoveL pPlace_App_3,v1000,fine,Ventosas3\WObj:=wobj0;
        MoveL pPlace_3,v1000,fine,Ventosas3\WObj:=wobj0;
        MoveL pPlace_App_3,v1000,fine,Ventosas3\WObj:=wobj0;
        MoveL Inicio_V3,v1000,fine,Ventosas3\WObj:=wobj0;
    ENDPROC
ENDMODULE

--- Controller Data/IRB120_3_58/SYSPAR/EIO.cfg ---
EIO:CFG_1.0:6:1::
#
EIO_SIGNAL:

      -Name "DO_Mover_C1" -SignalType "DO" -Label "Mover cinta 1"

      -Name "DO_Mover_C2" -SignalType "DO" -Label "Mover cinta 2"

      -Name "DO_Mover_C3" -SignalType "DO" -Label "Mover cinta 3"

      -Name "DO_Mover_C4" -SignalType "DO" -Label "Mover cinta 4"

      -Name "DO_Mover_C5" -SignalType "DO" -Label "Mover cinta 5"

      -Name "DO_Mover_C6" -SignalType "DO" -Label "Mover cinta 6"

      -Name "DO_Gen_C1_T1" -SignalType "DO"\
      -Label "Generador de cajas tipo 1 en la cinta 1"

      -Name "DO_Gen_C1_T2" -SignalType "DO"\
      -Label "Generador de cajas tipo 1 en la cinta 2"

      -Name "DO_Gen_C1_T3" -SignalType "DO"\
      -Label "Generador de cajas tipo 1 en la cinta 3"

      -Name "DO_Gen_C2_T1" -SignalType "DO"\
      -Label "Generador de cajas tipo 2 en la cinta 1"

      -Name "DO_Gen_C2_T2" -SignalType "DO"\
      -Label "Generador de cajas tipo 2 en la cinta 2"

      -Name "DO_Gen_C2_T3" -SignalType "DO"\
      -Label "Generador de cajas tipo 2 en la cinta 3"

      -Name "DO_Gen_C3_T1" -SignalType "DO"\
      -Label "Generador de cajas tipo 3 en la cinta 1"

      -Name "DO_Gen_C3_T2" -SignalType "DO"\
      -Label "Generador de cajas tipo 3 en la cinta 2"

      -Name "DO_Gen_C3_T3" -SignalType "DO"\
      -Label "Generador de cajas tipo 3 en la cinta 3"

      -Name "DI_Sen_C1_Bajo" -SignalType "DI"\
      -Label "Detectará los 3 tipos de cajas en la cinta 1"

      -Name "DI_Sen_C1_Medio" -SignalType "DI"\
      -Label "Detectará las cajas tipo 2 y 3 en la cinta 1"

      -Name "DI_Sen_C1_Alto" -SignalType "DI"\
      -Label "Detectará las cajas tipo 3 en la cinta 1"

      -Name "DI_Sen_C2_Bajo" -SignalType "DI"\
      -Label "Detectará los 3 tipos de cajas en la cinta 2"

      -Name "DI_Sen_C2_Medio" -SignalType "DI"\
      -Label "Detectará las cajas tipo 2 y 3 en la cinta 2"

      -Name "DI_Sen_C2_Alto" -SignalType "DI"\
      -Label "Detectará las cajas tipo 3 en la cinta 2"

      -Name "DI_Sen_C3_Bajo" -SignalType "DI"\
      -Label "Detectará los 3 tipos de cajas en la cinta 3"

      -Name "DI_Sen_C3_Medio" -SignalType "DI"\
      -Label "Detectará las cajas tipo 2 y 3 en la cinta 3"

      -Name "DI_Sen_C3_Alto" -SignalType "DI"\
      -Label "Detectará las cajas tipo 3 en la cinta 3"

      -Name "DO_Eliminar_Caja" -SignalType "DO"
